INTERFACE I_EventGroupItem EXTENDS I_Disposable

METHOD PUBLIC AddHandler
VAR_INPUT
	EventHandler : I_EventHandler;
END_VAR
END_METHOD

METHOD PUBLIC Emit
VAR_INPUT
	Event : I_Event;
END_VAR
END_METHOD

METHOD EqualTo : BOOL
VAR_INPUT
	Name : T_MAXSTRING;
END_VAR
END_METHOD

PROPERTY HasHandlers : BOOL
GET
END_GET
END_PROPERTY

PROPERTY PUBLIC Next : I_EventGroupItem
GET
END_GET
SET
END_SET
END_PROPERTY

PROPERTY PUBLIC Previous : I_EventGroupItem
GET
END_GET
SET
END_SET
END_PROPERTY

METHOD RemoveHandler
VAR_INPUT
	EventHandler : I_EventHandler;
END_VAR
END_METHOD

END_INTERFACE

(* stored: Version 1.1.0.1, ProductVersion 3.1.4024.12
   Itf I_EventGroupItem: Id {2467cd62-c253-0447-1c53-c19da17a624f}
   Method AddHandler: Id {20421c06-4630-028d-03f5-cd60b78124cb}
   Method Emit: Id {8b0adcf7-e892-0402-1da4-290b2049a4bf}
   Method EqualTo: Id {93db26b0-a3d1-098c-3ab9-a912cc48735c}
   Property HasHandlers: Id {22575985-e804-03a1-0e4d-4a73dca19d7d}
   Get Get: Id {04a62d7a-5100-0d7b-3877-5cd819b784cd}
   Property Next: Id {25e3ac2d-140c-0ec4-26d2-1a2babd80830}
   Get Get: Id {357f68df-9d2d-0bb5-2998-b1cb41f1c60e}
   Set Set: Id {1cda97b5-1714-0b75-074d-32a1a22899ec}
   Property Previous: Id {d42e328d-5300-0f71-03be-a2fa6ba651a0}
   Get Get: Id {6dfe0710-43fd-01ad-1179-738603cda23d}
   Set Set: Id {5d36066a-03bd-0d69-11a0-7b6e8440ea75}
   Method RemoveHandler: Id {4dc8b8c9-9725-0471-1f9e-b993618b1edb} *)
